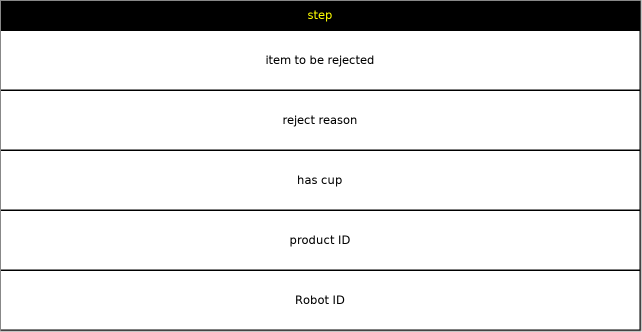
VISUALIZATION TWISTED_CUPS_SHIFT_ELEMENT_DESCRIPTION  // 642x332
    Rectangle (0,0 640x30), "step"
    Rectangle (0,30 640x60), "item to be rejected"
    Rectangle (0,90 640x60), "reject reason"
    Rectangle (0,150 640x60), "has cup"
    Rectangle (0,210 640x60), "product ID"
    Rectangle (0,270 640x60), "Robot ID"
END_VISUALIZATION

(* stored: Version 1.1.0.1, ProductVersion 3.1.4024.3
   Visu TWISTED_CUPS_SHIFT_ELEMENT_DESCRIPTION: Id {e29382c7-6840-407d-a3c6-49261e3b1f47} *)
